FUNCTION_BLOCK FB_SAFETY_AutoGroupErrACK
VAR_IN_OUT
	stSAFETYGroupIO: ST_SAFETYGroupIO;
END_VAR

stSAFETYGroupIO.ERR_Ack := stSAFETYGroupIO.FB_ERR OR stSAFETYGroupIO.COM_ERR OR stSAFETYGroupIO.OUT_ERR;

END_FUNCTION_BLOCK

(* stored: Version 1.1.0.1, ProductVersion 3.1.4022.12
   POU FB_SAFETY_AutoGroupErrACK: Id {3214460b-c5ea-4780-bf9a-c123c9c2f3e6}, SpecialFunc None *)
